Fanuc KAREL source: IO0084.KL

-- PROVISIONAL review KL for V1013-1; original PC SHA256 b896562a0a8b0722ab000618d1731a8bc5abba8f7ddb3573439f10c7b94f8f23
-- Incomplete behavior may be omitted. Consult companion uncertainty JSON. Do not deploy.
PROGRAM IO0084
%NOLOCKGROUP
-- UNRESOLVED_LOCAL_POOL 5 cells at code offset 13; source declarations unknown
-- DIRECT_LOCAL_WORD_ACCESS alone does not prove INTEGER, REAL, or BOOLEAN
BEGIN
  -- UNRESOLVED_PC offsets 0-18; opcodes 2B,2C,7B
  -- UNRESOLVED_PC offsets 23-30; opcodes 9D,23
  -- UNRESOLVED_PC offsets 35-49; opcodes 2E,22,9D,33,35
  -- UNRESOLVED_PC offsets 54-61; opcodes 9D,23
  -- UNRESOLVED_PC offsets 66-77; opcodes 2E,23
  -- UNRESOLVED_PC offsets 82-97; opcodes 21,19,64,23
  -- UNRESOLVED_PC offsets 102-106; opcodes 7F
  -- UNRESOLVED_PC offsets 111-115; opcodes 27,AA
  -- UNRESOLVED_PC offsets 120-124; opcodes 7F
END IO0084
